{attribute 'qualified_only'}
VAR_GLOBAL
	MainJibPistVelocity : LREAL;
	MainJibPistPosition : LREAL;
END_VAR

(* stored: Version 1.1.0.1, ProductVersion 3.1.4024.9
   GVL FromUnreal: Id {cce88e26-12dc-46fb-8614-84d84fcb5080} *)
